// TIA Portal project "2022.06.10_标准模拟量输入" (V17)

(* hardware
DEVICE "S7-1200 station_1"  S7-1200 Station
   slot 0: "Rack_0"  S7-1200 Rack  Rack  V1.0
   slot 1: "PLC_1"  CPU 1212C DC/DC/DC  6ES7 212-1AE40-0XB0  V4.5
   slot 2: "AI 4xRTD_1"  SM 1231 AI4 x RTD  6ES7 231-5PD32-0XB0  V2.0
*)

// ===== PLC "PLC_1"  CPU 1212C DC/DC/DC =====

VAR_GLOBAL   // PLC tag table "默认变量表"
   "通道0模拟值" AT %IW96 : Word;
   "百分比" AT %MD40 : DWord;
   "实际工程值" AT %MD44 : UDInt;
END_VAR

ORGANIZATION_BLOCK "Main"   // OB1, LAD, ProgramCycle
TITLE = "Main Program Sweep (Cycle)"
{ S7_Optimized_Access := 'TRUE' }
VERSION : 0.1
   VAR_INPUT
      Initial_Call : Bool;   // Initial call of this OB
      Remanence : Bool;   // =True, if remanent data are available
   END_VAR
BEGIN

REGION Network 1
   // 通道0接0-20ma电流信号，通道地址是iw96，对应实际工程中的0-50mpa，将0-27648转换成百分比输出
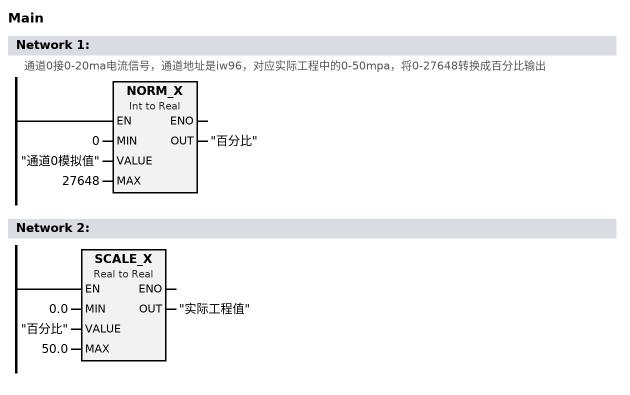
   RUNG wire#powerrail
      { S7_Templates := "[SrcType := Int, DestType := Real]" } Normalize(min := 0, value := "通道0模拟值", max := 27648, out => "百分比")
   END_RUNG
   // the same network as SCL:
   "百分比" := NORM_X(MIN := 0, VALUE := "通道0模拟值", MAX := 27648);
END_REGION

REGION Network 2
   RUNG wire#powerrail
      { S7_Templates := "[SrcType := Real, DestType := Real]" } Scale(min := 0.0, value := "百分比", max := 50.0, out => "实际工程值")
   END_RUNG
   // the same network as SCL:
   "实际工程值" := SCALE_X(MIN := 0.0, VALUE := "百分比", MAX := 50.0);
END_REGION
END_ORGANIZATION_BLOCK